// TIA Portal V20 export
DATA_BLOCK "Instance_FB_IO_Device_DB"   // DB104
// stored: AutoNumber false, InstanceOfName FB_IO_Device, InstanceOfType FB
"FB_IO_Device"
   // VAR_INPUT
   //    Life_Trigger : Bool;
   //    Emergency_Stop_Release : Bool;
   //    Trigger_Read_Serial_Number_Entrace_Functional_Test : Bool;
   //    Trigger_Read_Serial_Number_Exit_Functional_Test : Bool;
   //    Selected_Voltage_220V : Bool;
   //    Selected_Voltage_127V : Bool;
   //    Carousel_Frequency_Inverter_Fail : Bool;
   //    Conveyor_Belt_Functional_Test_Inverter_Fail : Bool;
   //    In : "IO_Device_Inputs";
   // END_VAR
   // VAR_OUTPUT
   //    Start : Bool;
   //    Manual_Turn_On_Motor_Caroussel : Bool;
   //    Manual_Turn_On_Motor_Conveyor_Belt : Bool;
   //    Water_Foutain_Fail_Functional_Test : Bool;
   //    Select_Motor_Speed : SInt;
   //    Carousel_Voltage_Selection : SInt;
   //    Out : "IO_Device_Outputs";
   // END_VAR
BEGIN
END_DATA_BLOCK
